{region '#Template'}
	{attribute 'Version' := '5.0.0.0'}
	{attribute 'Tags' := '"LCID": "1031", "Text": "AC, Setpoint, Temperatur, Cascade control"'}
	{attribute 'Tags' := '"LCID": "1033", "Text": "AC, Setpoint, Temperatur, Cascade control"'}
	{attribute 'Using' := '"Type": "Template", "URI": "BA2_Param"'}
	{attribute 'Description' := '"LCID": "1031", "Text": "Temperatur Kaskadenregelung"'}
	{attribute 'Description' := '"LCID": "1033", "Text": "Temperature Cascade control"'}
{endregion}
FUNCTION_BLOCK FB_BA_AC_TCasCtrl_01 EXTENDS FB_BA_View
VAR_INPUT
	fSpTRm					: REAL;
	fTRm					: REAL;
	stCmd					: ST_BA_Mdlt;						
END_VAR                                                         	
VAR_OUTPUT                                                      	
	fSpHtg					: REAL;
	fSpCol					: REAL;
	fSpErc					: REAL;
	fMax					: REAL;
	fMin					: REAL;
	bOn						: BOOL;	
END_VAR
VAR_INPUT CONSTANT
	SpHtg					: FB_BA_AV_Op;									
	SpCol					: FB_BA_AV_Op;																				  
	SpErc					: FB_BA_AV_Op;		
	Ctrl					: FB_BA_Loop;	
END_VAR
VAR
	PrioSwiVal				: FB_BA_PrioSwi_UDI04;	
	MuxCmd					: FB_BA_MMUX_B04;	

	MuxSpHtg				: FB_BA_MMUX_R04;
	MuxSpCol				: FB_BA_MMUX_R04;
	MuxSpErc				: FB_BA_MMUX_R04;
END_VAR
VAR // added by the converter: edge detectors and wires of the graphical bodies
    _w1 : ANY;
END_VAR

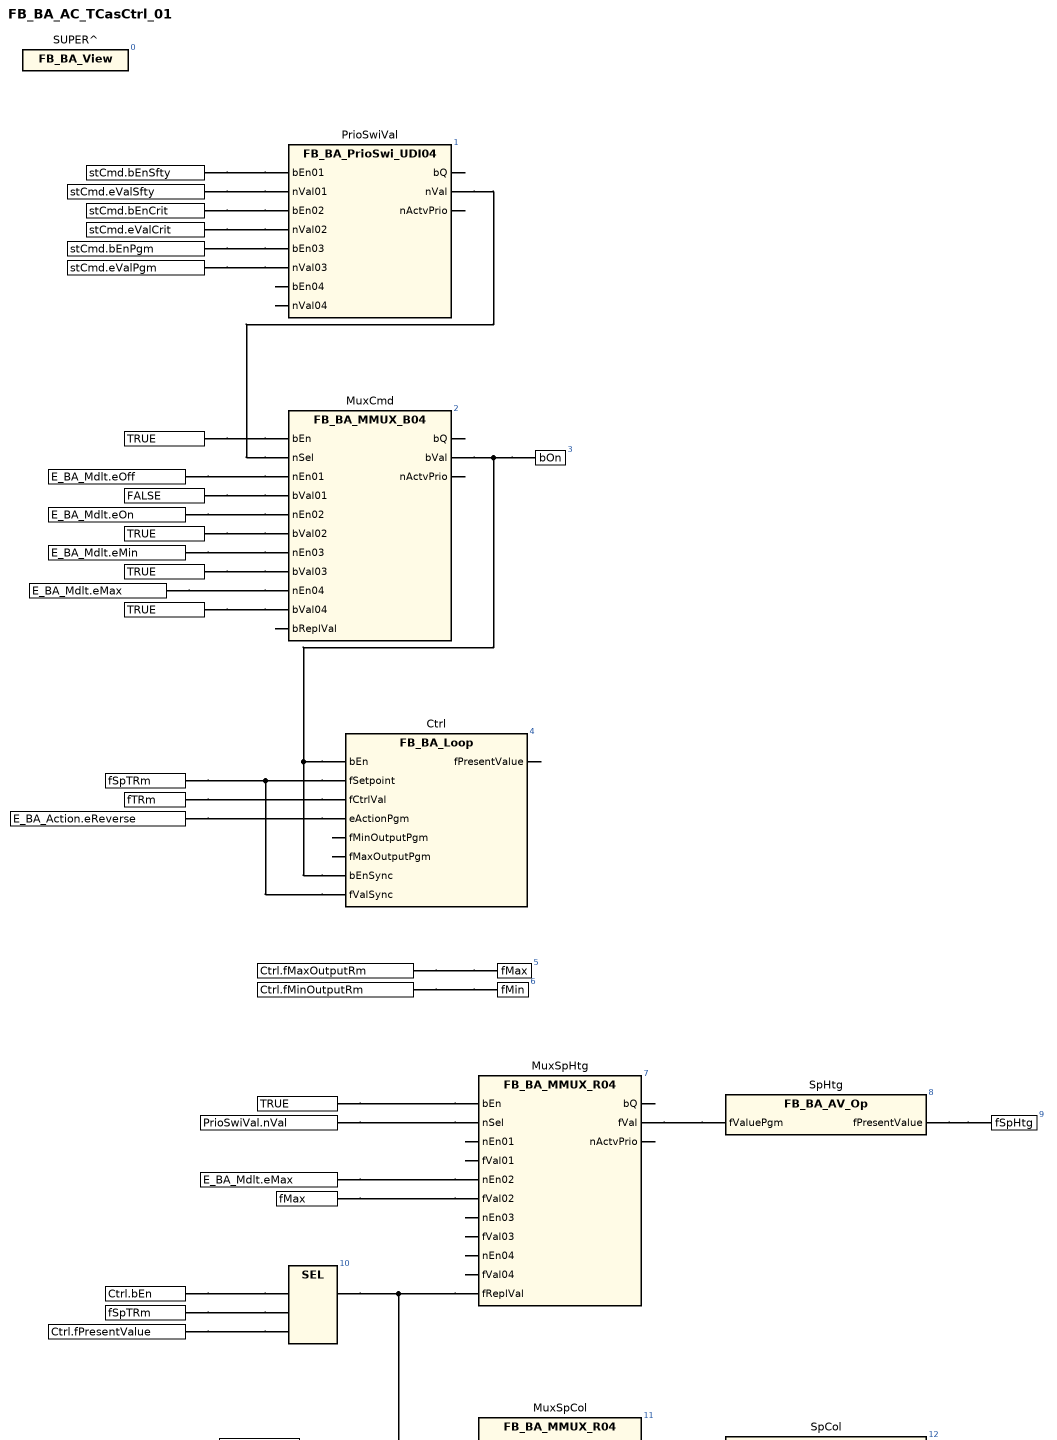
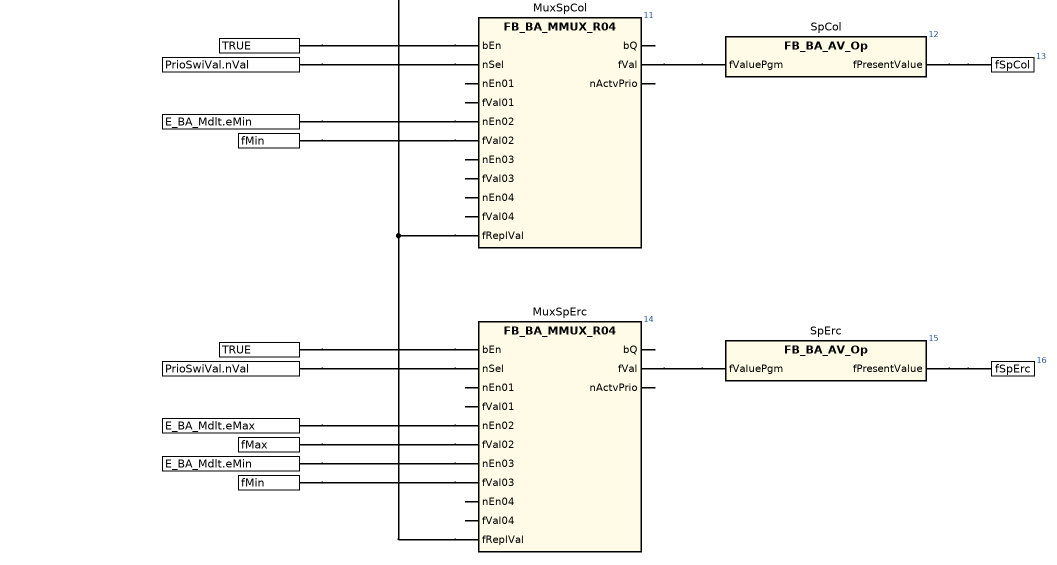
SUPER^(); // FB_BA_View
PrioSwiVal(
    bEn01 := stCmd.bEnSfty,
    nVal01 := stCmd.eValSfty,
    bEn02 := stCmd.bEnCrit,
    nVal02 := stCmd.eValCrit,
    bEn03 := stCmd.bEnPgm,
    nVal03 := stCmd.eValPgm); // FB_BA_PrioSwi_UDI04
MuxCmd(
    bEn := TRUE,
    nSel := PrioSwiVal.nVal,
    nEn01 := E_BA_Mdlt.eOff,
    bVal01 := FALSE,
    nEn02 := E_BA_Mdlt.eOn,
    bVal02 := TRUE,
    nEn03 := E_BA_Mdlt.eMin,
    bVal03 := TRUE,
    nEn04 := E_BA_Mdlt.eMax,
    bVal04 := TRUE); // FB_BA_MMUX_B04
bOn := MuxCmd.bVal;
Ctrl(
    bEn := MuxCmd.bVal,
    fSetpoint := fSpTRm,
    fCtrlVal := fTRm,
    eActionPgm := E_BA_Action.eReverse,
    bEnSync := MuxCmd.bVal,
    fValSync := fSpTRm); // FB_BA_Loop
fMax := Ctrl.fMaxOutputRm;
fMin := Ctrl.fMinOutputRm;
MuxSpHtg(bEn := TRUE, nSel := PrioSwiVal.nVal, nEn02 := E_BA_Mdlt.eMax, fVal02 := fMax, fReplVal := _w1); // FB_BA_MMUX_R04
SpHtg(fValuePgm := MuxSpHtg.fVal); // FB_BA_AV_Op
fSpHtg := SpHtg.fPresentValue;
_w1 := SEL(Ctrl.bEn, fSpTRm, Ctrl.fPresentValue);
MuxSpCol(bEn := TRUE, nSel := PrioSwiVal.nVal, nEn02 := E_BA_Mdlt.eMin, fVal02 := fMin, fReplVal := _w1); // FB_BA_MMUX_R04
SpCol(fValuePgm := MuxSpCol.fVal); // FB_BA_AV_Op
fSpCol := SpCol.fPresentValue;
MuxSpErc(
    bEn := TRUE,
    nSel := PrioSwiVal.nVal,
    nEn02 := E_BA_Mdlt.eMax,
    fVal02 := fMax,
    nEn03 := E_BA_Mdlt.eMin,
    fVal03 := fMin,
    fReplVal := _w1); // FB_BA_MMUX_R04
SpErc(fValuePgm := MuxSpErc.fVal); // FB_BA_AV_Op
fSpErc := SpErc.fPresentValue;

METHOD FB_init : BOOL
VAR_INPUT
	bInitRetains : BOOL; // if TRUE, the retain variables are initialized (warm start / cold start)
	bInCopyCode : BOOL;  // if TRUE, the instance afterwards gets moved into the copy code (online change)
END_VAR
SpHtg.iParent						:= THIS^;
SpHtg.iLabel						:= LblCtl_SuppyAirTempSetpointHeaterCalc; 				 	 
SpHtg.eUnit							:= E_BA_Unit.eTemperature_DegreesCelsius;  
SpHtg.fCOVIncrement					:= BA2_Param.fDefCOVIncrement;							

SpCol.iParent						:= THIS^;
SpCol.iLabel						:= LblCtl_SuppyAirTempSetpointCoolerCalc; 				 	 					 	 
SpCol.eUnit							:= E_BA_Unit.eTemperature_DegreesCelsius;  
SpCol.fCOVIncrement					:= BA2_Param.fDefCOVIncrement;							
									
SpErc.iParent						:= THIS^;
SpErc.iLabel						:= LblCtl_SuppyAirTempSetpointERCCalc; 									 	 
SpErc.eUnit							:= E_BA_Unit.eTemperature_DegreesCelsius;  
SpErc.fCOVIncrement					:= BA2_Param.fDefCOVIncrement;							

Ctrl.iParent						:= THIS^;
Ctrl.iLabel							:= LblFun_LoopObjectCascadeSupplyAirTemperature; 	
Ctrl.eOpMode						:= E_BA_PIDMode.ePID;							 	 										 
Ctrl.eOutputUnit					:= E_BA_Unit.eTemperature_DegreesCelsius;
Ctrl.fProportionalConstant			:= 1.5;
Ctrl.fIntegralConstant				:= 360;
Ctrl.fDerivativeConstant			:= 0;
Ctrl.fMaxOutputRm 					:= 32;
Ctrl.fMinOutputRm					:= 16;
Ctrl.fCOVIncrement					:= 0;
Ctrl.nDampConstant					:= 0;
Ctrl.fNeutralZone					:= 0;
END_METHOD

END_FUNCTION_BLOCK

(* stored: Version 1.1.0.1, ProductVersion 3.1.4024.12
   POU FB_BA_AC_TCasCtrl_01: Id {bc1a9304-2d21-4853-bfb6-7def207edbc7}, SpecialFunc None
   Method FB_init: Id {384a0b3e-897d-4d36-96e9-6ad8e9b68cda} *)
